{attribute 'qualified_only'}
{attribute 'strict'}
TYPE E_AxisParamCheckState :
(
    eInit,
    eSelect,
    eRead,
    eCheck,
    eAllParamValid,
    eInvalidParam
);
END_TYPE

(* stored: Version 1.1.0.1
   DUT E_AxisParamCheckState: Id {1344f39b-70f2-0dc2-3c34-7a926795d442} *)
